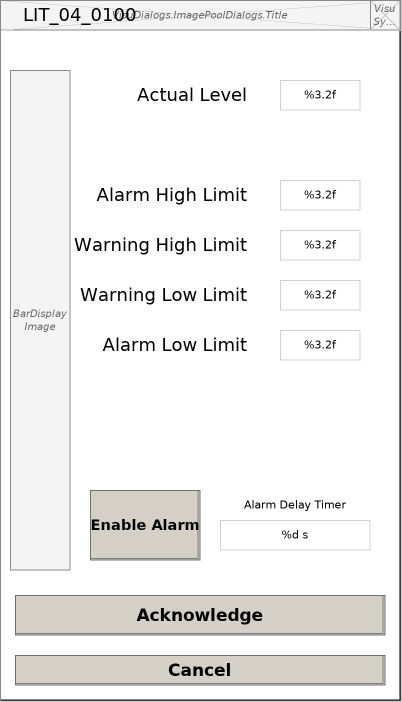
VISUALIZATION visuLITDiag  // 402x702
    Rectangle (0,0 400x700)
    Textfield (280,180 80x30), "%3.2f", text variable: progLITCntrl.LIT_04_0100.HHLimit
    Button (90,490 110x70), "Enable Alarm"
        toggle progHSVCntrl.HSV_04_0100.EnableAlarm
    Textfield (220,520 150x30), "%d s"
    Label (220,490 150x30), "Alarm Delay Timer"
    Image (0,0 400x30), image: VisuDialogs.ImagePoolDialogs.Title
    Group (370,0 30x30)
        RoundedRectangle (0,0 30x30)
        Image (0,0 30x30), image: VisuSymbols.Symbols.Wrong
    Button (15,655 370x30), "Cancel"
    Label (20,0 210x30), "LIT_04_0100"
    Label (0,180 250x30), "Alarm High Limit"
    Label (0,230 250x30), "Warning High Limit"
    Label (0,280 250x30), "Warning Low Limit"
    Label (0,330 250x30), "Alarm Low Limit"
    Textfield (280,230 80x30), "%3.2f", text variable: progLITCntrl.LIT_04_0100.HLimit
    Textfield (280,280 80x30), "%3.2f", text variable: progLITCntrl.LIT_04_0100.LLimit
    Textfield (280,330 80x30), "%3.2f", text variable: progLITCntrl.LIT_04_0100.LLLimit
    Button (15,595 370x40), "Acknowledge"
    Textfield (280,80 80x30), "%3.2f", text variable: progLITCntrl.LIT_04_0100.Level
    Label (0,80 250x30), "Actual Level"
    BarDisplayImage (10,70 60x500), value: progLITCntrl.LIT_04_0100.Level, style: BarDisplayImage-Gray, scale format: %.1f, scale 0..100
END_VISUALIZATION

(* stored: Version 1.1.0.1, ProductVersion 3.1.4022.17
   Visu visuLITDiag: Id {ab28e397-86b0-4cb0-a3d1-66ee0deb70e6} *)
